LIN {X 0,Y 121.787,Z 805.665,A -85,B 0,C 180,E1 2878.318,E2 2878.318} C_VEL
LIN {X 0,Y 116.097,Z 822.601,A -85,B 0,C 180,E1 2877.493,E2 2877.493} C_VEL
LIN {X 0,Y 108.657,Z 838.886,A -85,B 0,C 180,E1 2876.36,E2 2876.36} C_VEL
LIN {X 0,Y 99.908,Z 854.075,A -85,B 0,C 180,E1 2874.756,E2 2874.756} C_VEL
LIN {X 0,Y 89.778,Z 868.435,A -85,B 0,C 180,E1 2872.412,E2 2872.412} C_VEL
LIN {X 0,Y 78.455,Z 881.665,A -85,B 0,C 180,E1 2868.929,E2 2868.929} C_VEL
LIN {X 0,Y 66.631,Z 893.361,A -85,B 0,C 180,E1 2863.839,E2 2863.839} C_VEL
LIN {X 0,Y 54.791,Z 903.624,A -85,B 0,C 180,E1 2855.864,E2 2855.864} C_VEL
LIN {X 0,Y 43.914,Z 912.31,A -85,B 0,C 180,E1 2842.854,E2 2842.854} C_VEL
LIN {X 0,Y 36.024,Z 919.701,A -85,B 0,C 180,E1 2820.643,E2 2820.643} C_VEL
LIN {X 0,Y 35.208,Z 924.913,A -85,B 0,C 180,E1 2793.276,E2 2793.276} C_VEL
LIN {X 0,Y 35.853,Z 925.612,A -85,B 0,C 180,E1 2788.422,E2 2788.422} C_VEL
LIN {X 0,Y 36.537,Z 927.307,A -85,B 0,C 180,E1 2756.843,E2 2756.843} C_VEL
LIN {X 0,Y 45.825,Z 927.143,A -85,B 0,C 180,E1 2734.026,E2 2734.026} C_VEL
LIN {X 0,Y 60.619,Z 925.069,A -85,B 0,C 180,E1 2719.967,E2 2719.967} C_VEL
LIN {X 0,Y 77.65,Z 921.098,A -85,B 0,C 180,E1 2711.938,E2 2711.938} C_VEL
LIN {X 0,Y 93.765,Z 915.806,A -85,B 0,C 180,E1 2707.481,E2 2707.481} C_VEL
LIN {X 0,Y 110.307,Z 908.631,A -85,B 0,C 180,E1 2704.528,E2 2704.528} C_VEL
LIN {X 0,Y 120.349,Z 903.347,A -85,B 0,C 180,E1 2703.198,E2 2703.198} C_VEL
LIN {X 0,Y 119.208,Z 903.908,A -85,B 0,C 180,E1 2703.011,E2 2703.011} C_VEL
LIN {X 0,Y 111.364,Z 907.651,A -85,B 0,C 180,E1 2702.151,E2 2702.151} C_VEL
LIN {X 0,Y 95.466,Z 914.01,A -85,B 0,C 180,E1 2701.629,E2 2701.629} C_VEL
LIN {X 0,Y 85.897,Z 916.865,A -85,B 0,C 180,E1 2700.749,E2 2700.749} C_VEL
LIN {X 0,Y 81.817,Z 917.821,A -85,B 0,C 180,E1 2699.853,E2 2699.853} C_VEL
LIN {X 0,Y 66.284,Z 920.317,A -85,B 0,C 180,E1 2694.444,E2 2694.444} C_VEL
LIN {X 0,Y 50.664,Z 921.045,A -85,B 0,C 180,E1 2685.171,E2 2685.171} C_VEL
LIN {X 0,Y 37.361,Z 919.898,A -85,B 0,C 180,E1 2668.869,E2 2668.869} C_VEL
LIN {X 0,Y 29.581,Z 917,A -85,B 0,C 180,E1 2642.318,E2 2642.318} C_VEL
LIN {X 0,Y 30.031,Z 912.444,A -85,B 0,C 180,E1 2609.977,E2 2609.977} C_VEL
LIN {X 0,Y 38.083,Z 906.061,A -85,B 0,C 180,E1 2585.143,E2 2585.143} C_VEL
LIN {X 0,Y 49.337,Z 898.177,A -85,B 0,C 180,E1 2571.065,E2 2571.065} C_VEL
LIN {X 0,Y 62.239,Z 888.131,A -85,B 0,C 180,E1 2562.344,E2 2562.344} C_VEL
LIN {X 0,Y 74.086,Z 877.344,A -85,B 0,C 180,E1 2557.217,E2 2557.217} C_VEL
LIN {X 0,Y 85.317,Z 865.051,A -85,B 0,C 180,E1 2553.68,E2 2553.68} C_VEL
LIN {X 0,Y 95.758,Z 851.221,A -85,B 0,C 180,E1 2551.101,E2 2551.101} C_VEL
LIN {X 0,Y 104.857,Z 836.363,A -85,B 0,C 180,E1 2549.245,E2 2549.245} C_VEL
LIN {X 0,Y 112.532,Z 820.301,A -85,B 0,C 180,E1 2547.859,E2 2547.859} C_VEL
LIN {X 0,Y 118.512,Z 803.764,A -85,B 0,C 180,E1 2546.847,E2 2546.847} C_VEL
LIN {X 0,Y 122.737,Z 786.777,A -85,B 0,C 180,E1 2546.117,E2 2546.117} C_VEL
LIN {X 0,Y 126.017,Z 763.649,A -85,B 0,C 180,E1 2545.483,E2 2545.483} C_VEL
LIN {X 0,Y 132.223,Z 712.743,A -85,B 0,C 180,E1 2544.577,E2 2544.577} C_VEL
LIN {X 0,Y 131.726,Z 709.366,A -85,B 0,C 180,E1 2541.485,E2 2541.485} C_VEL
LIN {X 0,Y 131.509,Z 707.516,A -85,B 0,C 180,E1 2539.083,E2 2539.083} C_VEL
LIN {X 0,Y 131.449,Z 706.114,A -85,B 0,C 180,E1 2535.441,E2 2535.441} C_VEL
LIN {X 0,Y 131.773,Z 706.666,A -85,B 0,C 180,E1 2530.715,E2 2530.715} C_VEL
LIN {X 0,Y 132.269,Z 708.599,A -85,B 0,C 180,E1 2527.603,E2 2527.603} C_VEL
LIN {X 0,Y 133.016,Z 711.581,A -85,B 0,C 180,E1 2524.528,E2 2524.528} C_VEL
LIN {X 0,Y 133.166,Z 712.587,A -85,B 0,C 180,E1 2523.903,E2 2523.903} C_VEL
LIN {X 0,Y 124.043,Z 786.674,A -85,B 0,C 180,E1 2522.538,E2 2522.538} C_VEL
LIN {X 0,Y 119.886,Z 804.827,A -85,B 0,C 180,E1 2522.006,E2 2522.006} C_VEL
LIN {X 0,Y 114.342,Z 821.195,A -85,B 0,C 180,E1 2521.371,E2 2521.371} C_VEL
LIN {X 0,Y 106.992,Z 837.222,A -85,B 0,C 180,E1 2520.523,E2 2520.523} C_VEL
LIN {X 0,Y 97.998,Z 852.648,A -85,B 0,C 180,E1 2519.258,E2 2519.258} C_VEL
LIN {X 0,Y 87.55,Z 867.153,A -85,B 0,C 180,E1 2517.383,E2 2517.383} C_VEL
LIN {X 0,Y 75.838,Z 880.412,A -85,B 0,C 180,E1 2514.551,E2 2514.551} C_VEL
LIN {X 0,Y 62.935,Z 892.557,A -85,B 0,C 180,E1 2510.099,E2 2510.099} C_VEL
LIN {X 0,Y 50.197,Z 902.762,A -85,B 0,C 180,E1 2502.989,E2 2502.989} C_VEL
LIN {X 0,Y 37.989,Z 911.393,A -85,B 0,C 180,E1 2490.319,E2 2490.319} C_VEL
LIN {X 0,Y 28.709,Z 918.481,A -85,B 0,C 180,E1 2466.331,E2 2466.331} C_VEL
LIN {X 0,Y 27.25,Z 923.619,A -85,B 0,C 180,E1 2432.128,E2 2432.128} C_VEL
LIN {X 0,Y 27.734,Z 924.105,A -85,B 0,C 180,E1 2427.959,E2 2427.959} C_VEL
LIN {X 0,Y 29.593,Z 925.877,A -85,B 0,C 180,E1 2390.097,E2 2390.097} C_VEL
LIN {X 0,Y 41.793,Z 925.882,A -85,B 0,C 180,E1 2364.668,E2 2364.668} C_VEL
LIN {X 0,Y 57.406,Z 924.152,A -85,B 0,C 180,E1 2352.822,E2 2352.822} C_VEL
LIN {X 0,Y 74.438,Z 920.642,A -85,B 0,C 180,E1 2346.425,E2 2346.425} C_VEL
LIN {X 0,Y 92.66,Z 915.106,A -85,B 0,C 180,E1 2342.544,E2 2342.544} C_VEL
LIN {X 0,Y 81.817,Z 917.821,A -85,B 0,C 180,E1 2339.853,E2 2339.853} C_VEL
LIN {X 0,Y 74.464,Z 919.366,A -85,B 0,C 180,E1 2338.404,E2 2338.404} C_VEL
LIN {X 0,Y 57.392,Z 921.849,A -85,B 0,C 180,E1 2336.868,E2 2336.868} C_VEL
LIN {X 0,Y 49.319,Z 922.278,A -85,B 0,C 180,E1 2334.701,E2 2334.701} C_VEL
LIN {X 0,Y 47.295,Z 922.257,A -85,B 0,C 180,E1 2333.62,E2 2333.62} C_VEL
LIN {X 0,Y 32.149,Z 921.055,A -85,B 0,C 180,E1 2318.838,E2 2318.838} C_VEL
LIN {X 0,Y 22.192,Z 918.132,A -85,B 0,C 180,E1 2289.062,E2 2289.062} C_VEL
LIN {X 0,Y 22.422,Z 913.49,A -85,B 0,C 180,E1 2244.852,E2 2244.852} C_VEL
LIN {X 0,Y 32.339,Z 907.066,A -85,B 0,C 180,E1 2216.162,E2 2216.162} C_VEL
LIN {X 0,Y 45.063,Z 899.134,A -85,B 0,C 180,E1 2202.911,E2 2202.911} C_VEL
LIN {X 0,Y 58.952,Z 889.059,A -85,B 0,C 180,E1 2195.488,E2 2195.488} C_VEL
LIN {X 0,Y 71.399,Z 878.247,A -85,B 0,C 180,E1 2191.315,E2 2191.315} C_VEL
LIN {X 0,Y 83.049,Z 865.931,A -85,B 0,C 180,E1 2188.485,E2 2188.485} C_VEL
LIN {X 0,Y 93.8,Z 852.089,A -85,B 0,C 180,E1 2186.434,E2 2186.434} C_VEL
LIN {X 0,Y 103.122,Z 837.234,A -85,B 0,C 180,E1 2184.96,E2 2184.96} C_VEL
LIN {X 0,Y 110.968,Z 821.184,A -85,B 0,C 180,E1 2183.853,E2 2183.853} C_VEL
LIN {X 0,Y 117.072,Z 804.684,A -85,B 0,C 180,E1 2183.034,E2 2183.034} C_VEL
LIN {X 0,Y 121.42,Z 787.706,A -85,B 0,C 180,E1 2182.427,E2 2182.427} C_VEL
LIN {X 0,Y 124.679,Z 765.541,A -85,B 0,C 180,E1 2181.898,E2 2181.898} C_VEL
LIN {X 0,Y 130.611,Z 717.547,A -85,B 0,C 180,E1 2181.157,E2 2181.157} C_VEL
LIN {X 0,Y 130.427,Z 715.159,A -85,B 0,C 180,E1 2178.084,E2 2178.084} C_VEL
LIN {X 0,Y 130.457,Z 714.044,A -85,B 0,C 180,E1 2175.048,E2 2175.048} C_VEL
LIN {X 0,Y 130.696,Z 714.51,A -85,B 0,C 180,E1 2171.25,E2 2171.25} C_VEL
LIN {X 0,Y 131.076,Z 716.387,A -85,B 0,C 180,E1 2168.334,E2 2168.334} C_VEL
LIN {X 0,Y 131.264,Z 717.412,A -85,B 0,C 180,E1 2167.248,E2 2167.248} C_VEL
LIN {X 0,Y 122.575,Z 786.267,A -85,B 0,C 180,E1 2166.195,E2 2166.195} C_VEL
LIN {X 0,Y 118.274,Z 804.61,A -85,B 0,C 180,E1 2165.777,E2 2165.777} C_VEL
LIN {X 0,Y 112.468,Z 821.283,A -85,B 0,C 180,E1 2165.303,E2 2165.303} C_VEL
LIN {X 0,Y 104.841,Z 837.422,A -85,B 0,C 180,E1 2164.698,E2 2164.698} C_VEL
LIN {X 0,Y 95.7,Z 852.657,A -85,B 0,C 180,E1 2163.796,E2 2163.796} C_VEL
LIN {X 0,Y 85.069,Z 866.934,A -85,B 0,C 180,E1 2162.433,E2 2162.433} C_VEL
LIN {X 0,Y 72.997,Z 880.1,A -85,B 0,C 180,E1 2160.307,E2 2160.307} C_VEL
LIN {X 0,Y 60.078,Z 891.73,A -85,B 0,C 180,E1 2157.045,E2 2157.045} C_VEL
LIN {X 0,Y 46.423,Z 901.954,A -85,B 0,C 180,E1 2151.331,E2 2151.331} C_VEL
LIN {X 0,Y 32.933,Z 910.474,A -85,B 0,C 180,E1 2140.297,E2 2140.297} C_VEL
LIN {X 0,Y 21.528,Z 917.512,A -85,B 0,C 180,E1 2114.2,E2 2114.2} C_VEL
LIN {X 0,Y 19.631,Z 922.633,A -85,B 0,C 180,E1 2066.592,E2 2066.592} C_VEL
LIN {X 0,Y 23.908,Z 924.492,A -85,B 0,C 180,E1 2017.436,E2 2017.436} C_VEL
LIN {X 0,Y 39.088,Z 924.618,A -85,B 0,C 180,E1 1993.682,E2 1993.682} C_VEL
LIN {X 0,Y 57.135,Z 922.9,A -85,B 0,C 180,E1 1984.292,E2 1984.292} C_VEL
LIN {X 0,Y 65.899,Z 921.404,A -85,B 0,C 180,E1 1981.737,E2 1981.737} C_VEL
LIN {X 0,Y 50.146,Z 922.297,A -85,B 0,C 180,E1 1975.28,E2 1975.28} C_VEL
LIN {X 0,Y 47.295,Z 922.257,A -85,B 0,C 180,E1 1973.62,E2 1973.62} C_VEL
LIN {X 0,Y 40.067,Z 922.125,A -85,B 0,C 180,E1 1969.864,E2 1969.864} C_VEL
LIN {X 0,Y 25.028,Z 921.202,A -85,B 0,C 180,E1 1962.028,E2 1962.028} C_VEL
LIN {X 0,Y 16.974,Z 919.792,A -85,B 0,C 180,E1 1948.71,E2 1948.71} C_VEL
LIN {X 0,Y 15.252,Z 919.189,A -85,B 0,C 180,E1 1941.224,E2 1941.224} C_VEL
LIN {X 0,Y 15.75,Z 914.188,A -85,B 0,C 180,E1 1871.448,E2 1871.448} C_VEL
LIN {X 0,Y 27.707,Z 908.071,A -85,B 0,C 180,E1 1843.77,E2 1843.77} C_VEL
LIN {X 0,Y 41.926,Z 900.06,A -85,B 0,C 180,E1 1833.268,E2 1833.268} C_VEL
LIN {X 0,Y 56.601,Z 889.988,A -85,B 0,C 180,E1 1827.946,E2 1827.946} C_VEL
LIN {X 0,Y 69.524,Z 879.148,A -85,B 0,C 180,E1 1825.023,E2 1825.023} C_VEL
LIN {X 0,Y 81.499,Z 866.812,A -85,B 0,C 180,E1 1823.045,E2 1823.045} C_VEL
LIN {X 0,Y 92.488,Z 852.959,A -85,B 0,C 180,E1 1821.602,E2 1821.602} C_VEL
LIN {X 0,Y 101.983,Z 838.104,A -85,B 0,C 180,E1 1820.555,E2 1820.555} C_VEL
LIN {X 0,Y 109.959,Z 822.071,A -85,B 0,C 180,E1 1819.753,E2 1819.753} C_VEL
LIN {X 0,Y 116.137,Z 805.679,A -85,B 0,C 180,E1 1819.147,E2 1819.147} C_VEL
LIN {X 0,Y 120.615,Z 788.637,A -85,B 0,C 180,E1 1818.671,E2 1818.671} C_VEL
LIN {X 0,Y 123.866,Z 767.217,A -85,B 0,C 180,E1 1818.249,E2 1818.249} C_VEL
LIN {X 0,Y 129.397,Z 723.065,A -85,B 0,C 180,E1 1817.704,E2 1817.704} C_VEL
LIN {X 0,Y 129.462,Z 721.981,A -85,B 0,C 180,E1 1814.767,E2 1814.767} C_VEL
LIN {X 0,Y 129.645,Z 722.464,A -85,B 0,C 180,E1 1811.568,E2 1811.568} C_VEL
LIN {X 0,Y 129.701,Z 723.147,A -85,B 0,C 180,E1 1810.668,E2 1810.668} C_VEL
LIN {X 0,Y 121.666,Z 785.605,A -85,B 0,C 180,E1 1809.929,E2 1809.929} C_VEL
LIN {X 0,Y 117.331,Z 803.88,A -85,B 0,C 180,E1 1809.643,E2 1809.643} C_VEL
LIN {X 0,Y 111.472,Z 820.557,A -85,B 0,C 180,E1 1809.362,E2 1809.362} C_VEL
LIN {X 0,Y 103.78,Z 836.679,A -85,B 0,C 180,E1 1809.049,E2 1809.049} C_VEL
LIN {X 0,Y 94.267,Z 852.308,A -85,B 0,C 180,E1 1808.541,E2 1808.541} C_VEL
LIN {X 0,Y 83.765,Z 866.131,A -85,B 0,C 180,E1 1807.782,E2 1807.782} C_VEL
LIN {X 0,Y 71.459,Z 879.269,A -85,B 0,C 180,E1 1806.524,E2 1806.524} C_VEL
LIN {X 0,Y 58.183,Z 890.867,A -85,B 0,C 180,E1 1804.558,E2 1804.558} C_VEL
LIN {X 0,Y 44.009,Z 900.971,A -85,B 0,C 180,E1 1800.976,E2 1800.976} C_VEL
LIN {X 0,Y 29.204,Z 909.526,A -85,B 0,C 180,E1 1793.319,E2 1793.319} C_VEL
LIN {X 0,Y 15.138,Z 916.529,A -85,B 0,C 180,E1 1769.248,E2 1769.248} C_VEL
LIN {X 0,Y 11.549,Z 921.107,A -85,B 0,C 180,E1 1703.34,E2 1703.34} C_VEL
LIN {X 0,Y 20.887,Z 923.148,A -85,B 0,C 180,E1 1636.919,E2 1636.919} C_VEL
LIN {X 0,Y 38.987,Z 923.316,A -85,B 0,C 180,E1 1621.145,E2 1621.145} C_VEL
LIN {X 0,Y 39.787,Z 923.272,A -85,B 0,C 180,E1 1620.688,E2 1620.688} C_VEL
LIN {X 0,Y 23.677,Z 921.429,A -85,B 0,C 180,E1 1606.087,E2 1606.087} C_VEL
LIN {X 0,Y 15.252,Z 919.189,A -85,B 0,C 180,E1 1581.224,E2 1581.224} C_VEL
LIN {X 0,Y 11.824,Z 917.432,A -85,B 0,C 180,E1 1552.148,E2 1552.148} C_VEL
LIN {X 0,Y 14.363,Z 913.739,A -85,B 0,C 180,E1 1487.826,E2 1487.826} C_VEL
LIN {X 0,Y 21.056,Z 910.784,A -85,B 0,C 180,E1 1470.776,E2 1470.776} C_VEL
LIN {X 0,Y 24.917,Z 908.993,A -85,B 0,C 180,E1 1467.473,E2 1467.473} C_VEL
LIN {X 0,Y 40.037,Z 901.019,A -85,B 0,C 180,E1 1462.447,E2 1462.447} C_VEL
LIN {X 0,Y 55.303,Z 890.891,A -85,B 0,C 180,E1 1459.9,E2 1459.9} C_VEL
LIN {X 0,Y 68.525,Z 880.023,A -85,B 0,C 180,E1 1458.465,E2 1458.465} C_VEL
LIN {X 0,Y 80.708,Z 867.671,A -85,B 0,C 180,E1 1457.447,E2 1457.447} C_VEL
LIN {X 0,Y 91.85,Z 853.811,A -85,B 0,C 180,E1 1456.666,E2 1456.666} C_VEL
LIN {X 0,Y 101.457,Z 838.959,A -85,B 0,C 180,E1 1456.076,E2 1456.076} C_VEL
LIN {X 0,Y 109.522,Z 822.943,A -85,B 0,C 180,E1 1455.599,E2 1455.599} C_VEL
LIN {X 0,Y 115.765,Z 806.598,A -85,B 0,C 180,E1 1455.213,E2 1455.213} C_VEL
LIN {X 0,Y 120.334,Z 789.534,A -85,B 0,C 180,E1 1454.882,E2 1454.882} C_VEL
LIN {X 0,Y 123.572,Z 768.727,A -85,B 0,C 180,E1 1454.564,E2 1454.564} C_VEL
LIN {X 0,Y 128.475,Z 729.931,A -85,B 0,C 180,E1 1454.17,E2 1454.17} C_VEL
LIN {X 0,Y 121.234,Z 785.176,A -85,B 0,C 180,E1 1453.701,E2 1453.701} C_VEL
LIN {X 0,Y 116.833,Z 803.488,A -85,B 0,C 180,E1 1453.552,E2 1453.552} C_VEL
LIN {X 0,Y 111.043,Z 819.83,A -85,B 0,C 180,E1 1453.473,E2 1453.473} C_VEL
LIN {X 0,Y 103.328,Z 835.934,A -85,B 0,C 180,E1 1453.463,E2 1453.463} C_VEL
LIN {X 0,Y 94.053,Z 851.125,A -85,B 0,C 180,E1 1453.403,E2 1453.403} C_VEL
LIN {X 0,Y 83.209,Z 865.329,A -85,B 0,C 180,E1 1453.25,E2 1453.25} C_VEL
LIN {X 0,Y 70.793,Z 878.437,A -85,B 0,C 180,E1 1452.934,E2 1452.934} C_VEL
LIN {X 0,Y 57.344,Z 890.002,A -85,B 0,C 180,E1 1452.433,E2 1452.433} C_VEL
LIN {X 0,Y 42.847,Z 900.056,A -85,B 0,C 180,E1 1451.394,E2 1451.394} C_VEL
LIN {X 0,Y 27.347,Z 908.573,A -85,B 0,C 180,E1 1449.061,E2 1449.061} C_VEL
LIN {X 0,Y 11.01,Z 915.533,A -85,B 0,C 180,E1 1439.747,E2 1439.747} C_VEL
LIN {X 0,Y 3.649,Z 919.544,A -85,B 0,C 180,E1 1325.943,E2 1325.943} C_VEL
LIN {X 0,Y 13.992,Z 921.207,A -85,B 0,C 180,E1 1258.196,E2 1258.196} C_VEL
LIN {X 0,Y 6.052,Z 916.929,A -85,B 0,C 180,E1 1150.586,E2 1150.586} C_VEL
LIN {X 0,Y 20.786,Z 910.822,A -85,B 0,C 180,E1 1109.964,E2 1109.964} C_VEL
LIN {X 0,Y 24.917,Z 908.993,A -85,B 0,C 180,E1 1107.473,E2 1107.473} C_VEL
LIN {X 0,Y 27.709,Z 910.801,A -85,B 0,C 180,E1 1106.182,E2 1106.182} C_VEL
LIN {X 0,Y 27.709,Z 1007,A -85,B 0,C 180,E1 1106.182,E2 1106.182} C_VEL
LIN {X 0,Y 27.709,Z 1007,A -85,B 0,C 180,E1 1106.182,E2 1106.182}

QRS_NEXT_CUT()

QRS_NEXT()
QRS_HOME()

END
